FUNCTION_BLOCK dummy (* Basic FB with empty ECC *)
  (* Standard: 61499-2 *)
  (* Version 1.0, 2025-12-19, franz *)
  PACKAGE OSCAT::Network;
  EC_STATES
    START; (* Initial State *)
  END_STATES
END_FUNCTION_BLOCK
